TYPE FB_ServoAchse_Endschalter :
STRUCT
	//Positive Drehrichtung
	pos AT %I* : BOOL;
	//Negative Drehrichtung
	neg AT %I* : BOOL;
END_STRUCT
END_TYPE

(* stored: Version 1.1.0.1, ProductVersion 3.1.4018.5
   DUT FB_ServoAchse_Endschalter: Id {19effc6a-a419-4cd0-adef-9608ca06868d} *)
